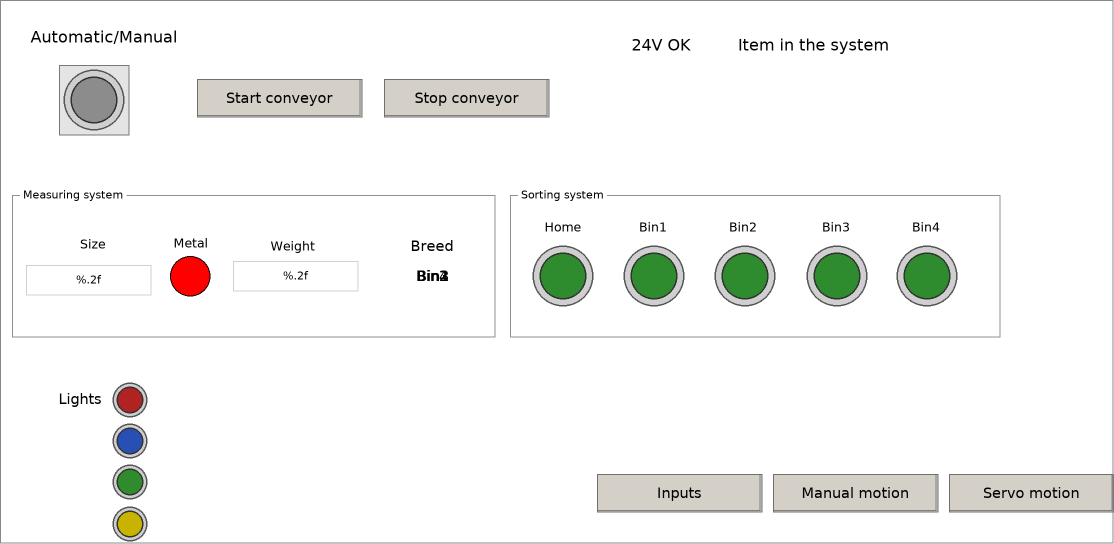
VISUALIZATION MainScreen  // 1114x544
    PushSwitch (59,65 70x70), variable: MeasuringData.AutomaticMode, behaviour: TOGGLE, style: Switch-PushSwitch-Gray
    Label (13,18 182x38), "Automatic/Manual"
    Button (197,79 165x38), "Start conveyor"
        OnMouseDown: execute { MeasuringData.StartConveyor := TRUE; }
        OnMouseUp: execute { MeasuringData.StartConveyor := FALSE; }
    Button (384,79 165x38), "Stop conveyor"
        OnMouseDown: execute { MeasuringData.StopConveyor := TRUE; }
        OnMouseUp: execute { MeasuringData.StopConveyor := FALSE; }
    Label (595,26 132x38), "24V OK", invisible if: MeasuringData.ControlSupplyOKOnHmi
    Label (729,26 169x38), "Item in the system", invisible if: MeasuringData.ItemInTheSystemOnHmi
    GroupBox (12,187 483x150), "Measuring system"
        Textfield (14,78 125x30), "%.2f", text variable: MeasuringData.SizeInCm
        Label (6,42 150x30), "Size"
        Ellipse (158,69 40x40), colour toggle: MeasuringData.MetalMaterial
        Label (138,41 82x30), "Metal"
        Textfield (221,74 125x30), "%.2f", text variable: MeasuringData.WeightInKg
        Label (240,44 82x30), "Weight"
        Label (379,44 82x30), "Breed"
        Label (380,74 82x30), "Bin1", invisible if: MeasuringData.Bin1BreedOnHmi
        Label (380,74 82x30), "Bin3", invisible if: MeasuringData.Bin3BreedOnHmi
        Label (379,74 82x30), "Bin4", invisible if: MeasuringData.Bin4BreedOnHmi
    GroupBox (510,187 490x150), "Sorting system"
        Lamp1 (18,54 70x70), variable: MeasuringData.TableAtHome, style: Lamp-Lamp1-Green
        Lamp1 (109,54 70x70), variable: MeasuringData.TableAtBin1, style: Lamp-Lamp1-Green
        Lamp1 (200,54 70x70), variable: MeasuringData.TableAtBin2, style: Lamp-Lamp1-Green
        Lamp1 (292,54 70x70), variable: MeasuringData.TableAtBin3, style: Lamp-Lamp1-Green
        Lamp1 (382,54 70x70), variable: MeasuringData.TableAtBin4, style: Lamp-Lamp1-Green
        Label (12,25 82x30), "Home"
        Label (102,25 82x30), "Bin1"
        Label (192,25 82x30), "Bin2"
        Label (285,25 82x30), "Bin3"
        Label (375,25 82x30), "Bin4"
    Button (597,474 165x38), "Inputs"
    Button (773,474 165x38), "Manual motion"
    Button (949,474 165x38), "Servo motion"
    Label (39,384 82x30), "Lights"
    Lamp1 (110,380 40x40), variable: Outputs.Red_light, style: Lamp-Lamp1-Red
    Lamp1 (110,421 40x40), variable: Outputs.Blue_light, style: Lamp-Lamp1-Blue
    Lamp1 (110,462 40x40), variable: Outputs.Green_light, style: Lamp-Lamp1-Green
    Lamp1 (110,504 40x40), variable: Outputs.Yellow_light, style: Lamp-Lamp1-Yellow
    Label (391,261 82x30), "Bin2", invisible if: MeasuringData.Bin2BreedOnHmi
END_VISUALIZATION

(* stored: Version 1.1.0.1, ProductVersion 3.1.4024.13
   Visu MainScreen: Id {677a8f57-d7ba-4c64-a33e-5830dd9e2f87} *)
